FUNCTION_BLOCK EA_2_leftSwitch
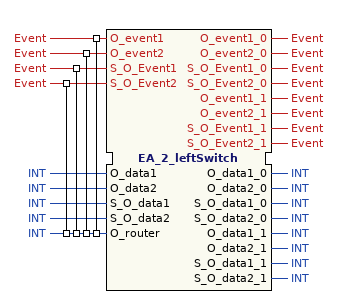
  EVENT_INPUT
    O_event1 WITH O_router;
    O_event2 WITH O_router;
    S_O_Event1 WITH O_router;
    S_O_Event2 WITH O_router;
  END_EVENT
  EVENT_OUTPUT
    O_event1_0;
    O_event2_0;
    S_O_Event1_0;
    S_O_Event2_0;
    O_event1_1;
    O_event2_1;
    S_O_Event1_1;
    S_O_Event2_1;
  END_EVENT
  VAR_INPUT
    O_data1 : INT;
    O_data2 : INT;
    S_O_data1 : INT;
    S_O_data2 : INT;
    O_router : INT;
  END_VAR
  VAR_OUTPUT
    O_data1_0 : INT;
    O_data2_0 : INT;
    S_O_data1_0 : INT;
    S_O_data2_0 : INT;
    O_data1_1 : INT;
    O_data2_1 : INT;
    S_O_data1_1 : INT;
    S_O_data2_1 : INT;
  END_VAR
  EC_STATES
    Start;
    O_event1_0_state : O_event1_0_algorithm -> O_event1_0;
    O_event2_0_state : O_event2_0_algorithm -> O_event2_0;
    S_O_Event1_0_state : S_O_Event1_0_algorithm -> S_O_Event1_0;
    S_O_Event2_0_state : S_O_Event2_0_algorithm -> S_O_Event2_0;
    O_event1_1_state : O_event1_1_algorithm -> O_event1_1;
    O_event2_1_state : O_event2_1_algorithm -> O_event2_1;
    S_O_Event1_1_state : S_O_Event1_1_algorithm -> S_O_Event1_1;
    S_O_Event2_1_state : S_O_Event2_1_algorithm -> S_O_Event2_1;
  END_STATES
  EC_TRANSITIONS
    O_event1_0_state TO Start := 1;
    Start TO O_event1_0_state := O_event1[O_router = 0];
    O_event2_0_state TO Start := 1;
    Start TO O_event2_0_state := O_event2[O_router = 0];
    S_O_Event1_0_state TO Start := 1;
    Start TO S_O_Event1_0_state := S_O_Event1[O_router = 0];
    S_O_Event2_0_state TO Start := 1;
    Start TO S_O_Event2_0_state := S_O_Event2[O_router = 0];
    O_event1_1_state TO Start := 1;
    Start TO O_event1_1_state := O_event1[O_router = 1];
    O_event2_1_state TO Start := 1;
    Start TO O_event2_1_state := O_event2[O_router = 1];
    S_O_Event1_1_state TO Start := 1;
    Start TO S_O_Event1_1_state := S_O_Event1[O_router = 1];
    S_O_Event2_1_state TO Start := 1;
    Start TO S_O_Event2_1_state := S_O_Event2[O_router = 1];
  END_TRANSITIONS
  ALGORITHM O_event1_0_algorithm IN ST:
O_data1_0 := O_data1;
O_data2_0 := O_data2;
S_O_data1_0 := S_O_data1;
S_O_data2_0 := S_O_data2;
  END_ALGORITHM
  ALGORITHM O_event2_0_algorithm IN ST:
O_data1_0 := O_data1;
O_data2_0 := O_data2;
S_O_data1_0 := S_O_data1;
S_O_data2_0 := S_O_data2;
  END_ALGORITHM
  ALGORITHM S_O_Event1_0_algorithm IN ST:
O_data1_0 := O_data1;
O_data2_0 := O_data2;
S_O_data1_0 := S_O_data1;
S_O_data2_0 := S_O_data2;
  END_ALGORITHM
  ALGORITHM S_O_Event2_0_algorithm IN ST:
O_data1_0 := O_data1;
O_data2_0 := O_data2;
S_O_data1_0 := S_O_data1;
S_O_data2_0 := S_O_data2;
  END_ALGORITHM
  ALGORITHM O_event1_1_algorithm IN ST:
O_data1_1 := O_data1;
O_data2_1 := O_data2;
S_O_data1_1 := S_O_data1;
S_O_data2_1 := S_O_data2;
  END_ALGORITHM
  ALGORITHM O_event2_1_algorithm IN ST:
O_data1_1 := O_data1;
O_data2_1 := O_data2;
S_O_data1_1 := S_O_data1;
S_O_data2_1 := S_O_data2;
  END_ALGORITHM
  ALGORITHM S_O_Event1_1_algorithm IN ST:
O_data1_1 := O_data1;
O_data2_1 := O_data2;
S_O_data1_1 := S_O_data1;
S_O_data2_1 := S_O_data2;
  END_ALGORITHM
  ALGORITHM S_O_Event2_1_algorithm IN ST:
O_data1_1 := O_data1;
O_data2_1 := O_data2;
S_O_data1_1 := S_O_data1;
S_O_data2_1 := S_O_data2;
  END_ALGORITHM
END_FUNCTION_BLOCK
